Omron CX-Programmer project NewProject (CX-Programmer 9.51)

# PLC my_first_project: CP1L L
; Myfristproject

## Global symbols (name address type ; comment)
W0.01 BOOL  ; comment

## Program NewProgram1 (cyclic task 0)
Local symbols
button_1 0.00 BOOL  ; comment
button_2 0.01 BOOL  ; comment
button_3 0.02 BOOL  ; comment
out_3 100.02 BOOL  ; comment

### Section Section1

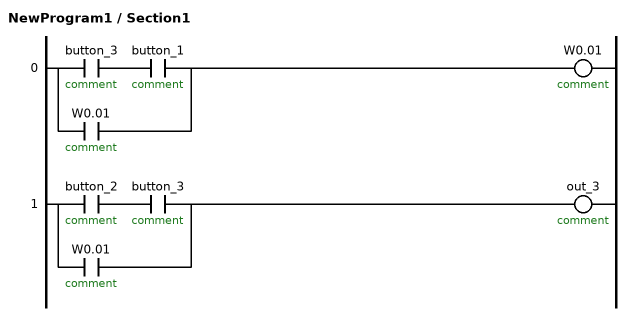
; rung 0
LD button_3  ; comment
AND button_1  ; comment
OR W0.01  ; comment
OUT W0.01  ; comment
; rung 1
LD button_2  ; comment
AND button_3  ; comment
OR W0.01  ; comment
OUT out_3  ; comment

### Section END
; rung 0
END(001)